FUNCTION_BLOCK DigitalLampWithPushButton_1 EXTENDS OnOffDevice
VAR
	IN AT%I* : BOOL;
	
	rtIN: R_TRIG;
END_VAR


	rtIN(CLK:= IN, Q=> );

	IF rtIN.Q THEN
		IF Status = TRUE THEN
			TurnOff();
		ELSE
			TurnOn();
		END_IF
	END_IF

END_FUNCTION_BLOCK

(* stored: Version 1.1.0.1, ProductVersion 3.1.4024.13
   POU DigitalLampWithPushButton_1: Id {ef09533f-2613-4a79-8bb5-783bb9f92126}, SpecialFunc None *)
